PROGRAM F_Faults
VAR

END_VAR

IF FIO.b_IN_1 AND GVL.bReset THEN 
	FIO.b_OUT_13 := TRUE;
ELSE
	FIO.b_OUT_13 := FALSE;
END_IF

END_PROGRAM

(* stored: Version 1.1.0.1
   POU F_Faults: Id {4e32251a-45ed-4bd7-b243-fab3917a6db3}, SpecialFunc None *)
